FUNCTION_BLOCK FB_CTU (* Up counter *)
  PACKAGE iec61131::counters;
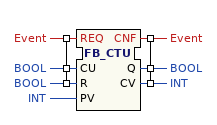
  EVENT_INPUT
    REQ WITH CU, R; (* Normal Execution Request *)
  END_EVENT
  EVENT_OUTPUT
    CNF WITH Q, CV; (* Execution Confirmation *)
  END_EVENT
  VAR_INPUT
    CU : BOOL; (* Count up *)
    R : BOOL; (* Reset *)
    PV : INT; (* Preset value *)
  END_VAR
  VAR_OUTPUT
    Q : BOOL; (* Output *)
    CV : INT; (* Count value *)
  END_VAR
  ALGORITHM REQ IN ST:
IF R THEN
  CV := 0;
ELSIF CU AND CV < 32767 THEN
  CV := CV + 1;
END_IF;
Q := CV>= PV;
  END_ALGORITHM
END_FUNCTION_BLOCK
